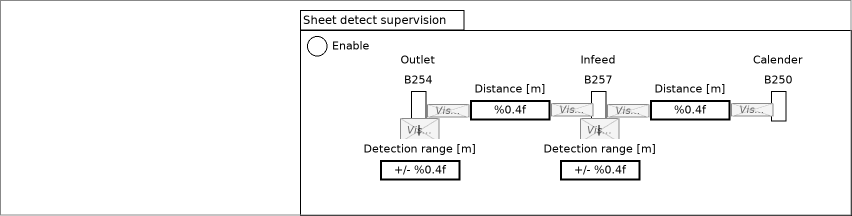
VISUALIZATION VISU_SheetDetectSupervision  // 852x216
VAR_IN_OUT
  mInst : FB_SheetDetectSupervision;
END_VAR
    Rectangle (300,10 164x20), "Sheet detect supervision"
    Rectangle (300,30 552x186)
    RoundedRectangle (771,91 15x30)
    Rectangle (756,70 45x20), "B250"
    RoundedRectangle (591,91 15x30)
    Rectangle (576,70 45x20), "B257"
    RoundedRectangle (411,91 15x30)
    Rectangle (396,70 45x20), "B254"
    Rectangle (650,100 80x20), "%0.4f", text variable: mInst.RemSheetDetectSupervisionPar.fR_SheetDetectDistance01
        OnMouseClick: write the text variable via Default
    Rectangle (650,79 80x20), "Distance [m]"
    Image (607,104 42x13), image: VisuSymbols.Symbols.ArrowBoldLeft
    Image (731,103 42x13), image: VisuSymbols.Symbols.ArrowBoldRight
    Rectangle (470,100 80x20), "%0.4f", text variable: mInst.RemSheetDetectSupervisionPar.fR_SheetDetectDistance02
        OnMouseClick: write the text variable via Default
    Rectangle (470,79 80x20), "Distance [m]"
    Image (427,104 42x13), image: VisuSymbols.Symbols.ArrowBoldLeft
    Image (551,103 42x13), image: VisuSymbols.Symbols.ArrowBoldRight
    Image (580,118 39x24), image: VisuSymbols.Symbols.DoubleArrow3
    Rectangle (560,160 80x20), "+/- %0.4f", text variable: mInst.RemSheetDetectSupervisionPar.fR_SheetDetectRange01_m
        OnMouseClick: write the text variable via Default
    Rectangle (540,139 120x20), "Detection range [m]"
    Line (599,135) (599,125)
    Rectangle (568,50 60x20), "Infeed"
    Rectangle (748,50 60x20), "Calender"
    Rectangle (388,50 60x20), "Outlet"
    Ellipse (307,36 20x20), tooltip "Reset"
        toggle mInst.RemSheetDetectSupervisionPar.bR_Enable
    Rectangle (329,36 60x20), "Enable"
    Image (400,118 39x24), image: VisuSymbols.Symbols.DoubleArrow3
    Rectangle (380,160 80x20), "+/- %0.4f", text variable: mInst.RemSheetDetectSupervisionPar.fR_SheetDetectRange02_m
        OnMouseClick: write the text variable via Default
    Rectangle (360,139 120x20), "Detection range [m]"
    Line (419,135) (419,125)
END_VISUALIZATION

(* stored: Version 1.1.0.1, ProductVersion 3.1.4024.11
   Visu VISU_SheetDetectSupervision: Id {b9958c72-9de1-48ab-a536-2073d9ffa3ff} *)
